// TwinCAT 3 PLC project PLC1
// ProgramVersion: 3.1.4026.13
// libraries:
//   Tc2_Standard, * (Beckhoff Automation GmbH)
//   Tc2_System, * (Beckhoff Automation GmbH)
//   Tc3_Module, * (Beckhoff Automation GmbH)
// project tree:
//   / GlobalTextList.TcGTLO (not stored), PlcTask.TcTTO (not stored)
//   GVLs/ Devices.TcGVL, GVL.TcGVL (not stored)
//   POUs/Devices/ FB_MotorContactor.TcPOU, FB_NormallyClosedPB.TcPOU (not stored), FB_NormallyClosedSensor.TcPOU (not stored), FB_NormallyOpenPB.TcPOU, FB_NormallyOpenSensor.TcPOU
//   POUs/ I_Pushbutton.TcIO, I_Sensor.TcIO, MAIN.TcPOU
//   POUs/Machine/ FB_ConveyorMachine.TcPOU (not stored)
// real-time tasks:
//   TASK PlcTask: cycle T#10ms, priority 20, ADS port 350

// ---- GVLs/Devices.TcGVL
VAR_GLOBAL
	//Conveyor A
	ConvA_Stop 				: FB_NormallyClosedPB;
	ConvA_EStop			 	: FB_NormallyClosedPB;
	ConvA_Start	 			: FB_NormallyOpenPB;
	ConvA_ProdDetect		: FB_NormallyOpenSensor;
	ConvA_ConvFull	 		: FB_NormallyOpenSensor;
	ConvA_Motor				: FB_MotorContactor;	
	                        
	//Conveyor B            
	ConvB_Stop 		   		: FB_NormallyOpenPB;
	ConvB_EStop		   	 	: FB_NormallyClosedPB;
	ConvB_Start	 	  		: FB_NormallyOpenPB;
	ConvB_ProdDetect		: FB_NormallyClosedSensor;
	ConvB_ConvFull	 	 	: FB_NormallyOpenSensor;
	ConvB_Motor				: FB_MotorContactor;
	                        
	//Conveyor C            
	ConvC_Stop 		   		: FB_NormallyClosedPB;
	ConvC_EStop		   	 	: FB_NormallyOpenPB;
	ConvC_Start	 	  		: FB_NormallyOpenPB;
	ConvC_ProdDetect	 	: FB_NormallyOpenSensor;
	ConvC_ConvFull	  		: FB_NormallyClosedSensor;
	ConvC_Motor				: FB_MotorContactor;	
	                        
	//Conveyor D            
	ConvD_Stop 		   		: FB_NormallyClosedPB;
	ConvD_EStop		   	 	: FB_NormallyClosedPB;
	ConvD_Start	 	  		: FB_NormallyOpenPB;
	ConvD_ProdDetect	 	: FB_NormallyOpenSensor;
	ConvD_ConvFull	  		: FB_NormallyOpenSensor;
	ConvD_Motor				: FB_MotorContactor;	
	                        
	//Conveyor E            
	ConvE_Stop 		   		: FB_NormallyClosedPB;
	ConvE_EStop		   	 	: FB_NormallyClosedPB;
	ConvE_Start	 	  		: FB_NormallyOpenPB;
	ConvE_ProdDetect	 	: FB_NormallyOpenSensor;
	ConvE_ConvFull	  		: FB_NormallyOpenSensor;
	ConvE_Motor				: FB_MotorContactor;
END_VAR

// ---- POUs/I_Pushbutton.TcIO
INTERFACE I_Pushbutton

PROPERTY IsPressed : BOOL
GET
END_GET
END_PROPERTY

PROPERTY IsReleased : BOOL
GET
END_GET
END_PROPERTY

END_INTERFACE

// ---- POUs/I_Sensor.TcIO
INTERFACE I_Sensor

PROPERTY IsActive : BOOL
GET
END_GET
END_PROPERTY

END_INTERFACE

// ---- POUs/Devices/FB_NormallyOpenPB.TcPOU
FUNCTION_BLOCK FB_NormallyOpenPB IMPLEMENTS I_Pushbutton
VAR
	Input AT %I* : BOOL;
END_VAR

PROPERTY IsPressed : BOOL
GET
IsPressed := Input;
END_GET
END_PROPERTY

PROPERTY IsReleased : BOOL
GET
IsReleased := NOT Input;
END_GET
END_PROPERTY

END_FUNCTION_BLOCK

// ---- POUs/Devices/FB_NormallyOpenSensor.TcPOU
FUNCTION_BLOCK FB_NormallyOpenSensor IMPLEMENTS I_Sensor
VAR
	Input AT %I* : BOOL;
END_VAR

PROPERTY IsActive : BOOL
GET
IsActive := Input;
END_GET
END_PROPERTY

END_FUNCTION_BLOCK

// ---- POUs/Devices/FB_MotorContactor.TcPOU
FUNCTION_BLOCK FB_MotorContactor 
VAR
	Output AT %Q* : BOOL;
END_VAR

METHOD SwitchOff : BOOL
VAR_INPUT
END_VAR
Output := FALSE;
END_METHOD

METHOD SwitchOn : BOOL
VAR_INPUT
END_VAR
Output := TRUE;
END_METHOD

END_FUNCTION_BLOCK

// ---- POUs/MAIN.TcPOU
PROGRAM MAIN
VAR
	ConvA : FB_ConveyorMachine(ConvA_Stop,ConvA_EStop, ConvA_Start, ConvA_ProdDetect,
							   ConvA_ConvFull, ConvA_Motor);

	ConvB : FB_ConveyorMachine(ConvB_Stop,ConvB_EStop, ConvB_Start, ConvB_ProdDetect,
							   ConvB_ConvFull, ConvB_Motor);
	
	ConvC : FB_ConveyorMachine(ConvC_Stop,ConvC_EStop, ConvC_Start, ConvC_ProdDetect,
							   ConvC_ConvFull, ConvC_Motor);	

	ConvD : FB_ConveyorMachine(ConvD_Stop,ConvD_EStop, ConvD_Start, ConvD_ProdDetect,
							   ConvD_ConvFull, ConvD_Motor);

	ConvE : FB_ConveyorMachine(ConvE_Stop,ConvE_EStop, ConvE_Start, ConvE_ProdDetect,
							   ConvE_ConvFull, ConvE_Motor);
END_VAR

ConvA();
ConvB();
ConvC();
ConvD();
ConvE();

END_PROGRAM
